FUNCTION_BLOCK VN_model
  (* Version 1.0, 2005-09-21, Goran Cengic, Chalmers *)
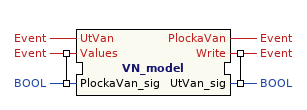
  EVENT_INPUT
    UtVan;
    Values WITH PlockaVan_sig;
  END_EVENT
  EVENT_OUTPUT
    PlockaVan;
    Write WITH UtVan_sig;
  END_EVENT
  VAR_INPUT
    PlockaVan_sig : BOOL;
  END_VAR
  VAR_OUTPUT
    UtVan_sig : BOOL;
  END_VAR
END_FUNCTION_BLOCK
